(* IEC 61131-3 sources: repolevel_ST_code_completion/output/0121完整版本/repoeval_electronic_cam_motion/readful_result_history, 4 files *)

(* ---- F_AxisStatusToString_0.st ---- *)
FUNCTION F_AxisStatusToString : STRING
VAR_INPUT
	fbReadStatus	:	MC_ReadStatus;		//轴状态读取功能块
END_VAR
IF fbReadStatus.Errorstop THEN
	F_AxisStatusToString := 'Errorstop';
	RETURN;
END_IF

IF fbReadStatus.Disabled THEN
	F_AxisStatusToString := 'Disabled';
	RETURN;
END_IF

IF fbReadStatus.Homing THEN
	F_AxisStatusToString := 'Homing';
	RETURN;
END_IF

IF fbReadStatus.Stopping THEN
	F_AxisStatusToString := 'Stopping';
	RETURN;
END_IF

IF fbReadStatus.SynchronizedMotion THEN
	F_AxisStatusToString := 'SynchronizedMotion';
	RETURN;
END_IF

IF fbReadStatus.ContinuousMotion THEN
	F_AxisStatusToString := 'ContinuousMotion';
	RETURN;
END_IF

IF fbReadStatus.Standstill THEN
	F_AxisStatusToString := 'Standstill';
	RETURN;
END_IF

F_AxisStatusToString := 'Unknown';
RETURN;
END_FUNCTION

(* ---- FB_DualAxisPower_0.st ---- *)
FUNCTION_BLOCK FB_DualAxisPower
VAR_INPUT
	Axis1			:	AXIS_REF;			//轴1引用
	Axis2			:	AXIS_REF;			//轴2引用
	bPowerOn		:	BOOL;				//电源使能信号
END_VAR
VAR_OUTPUT
	bPowerDone		:	BOOL;				//两轴都准备就绪
	bAxis1Ready		:	BOOL;				//轴1准备就绪
	bAxis2Ready		:	BOOL;				//轴2准备就绪
	bError			:	BOOL;				//错误标志
END_VAR
VAR
	fbPower1		:	MC_Power;			//轴1电源控制
	fbPower2		:	MC_Power;			//轴2电源控制
	bAxis1Error		:	BOOL;				//轴1错误标志
	bAxis2Error		:	BOOL;				//轴2错误标志
END_VAR

fbPower1(
	Axis := Axis1,
	Enable := TRUE,
	bDriveStart := bPowerOn,
	bRegulatorOn := bPowerOn
);

fbPower2(
	Axis := Axis2,
	Enable := TRUE,
	bDriveStart := bPowerOn,
	bRegulatorOn := bPowerOn
);

bAxis1Ready := fbPower1.Status = MC_POWER_STATUS_READY;
bAxis2Ready := fbPower2.Status = MC_POWER_STATUS_READY;

bAxis1Error := fbPower1.Error;
bAxis2Error := fbPower2.Error;

bError := bAxis1Error OR bAxis2Error;
bPowerDone := bAxis1Ready AND bAxis2Ready AND NOT bError;
END_FUNCTION_BLOCK

(* ---- FB_DualAxisReset_0.st ---- *)
FUNCTION_BLOCK FB_DualAxisReset
VAR_INPUT
	Axis1			:	AXIS_REF;			//轴1引用
	Axis2			:	AXIS_REF;			//轴2引用
	bExecute		:	BOOL;				//执行复位信号
END_VAR
VAR_OUTPUT
	bDone			:	BOOL;				//复位完成
	bBusy			:	BOOL;				//复位进行中
	bError			:	BOOL;				//错误标志
END_VAR
VAR
	fbReset1		:	MC_Reset;			//轴1复位
	fbReset2		:	MC_Reset;			//轴2复位
	fbReadStatus1	:	MC_ReadStatus;		//轴1状态读取
	fbReadStatus2	:	MC_ReadStatus;		//轴2状态读取
	bError1			:	BOOL;				//轴1错误标志
	bError2			:	BOOL;				//轴2错误标志
	nState			:	UDINT;				//状态机
END_VAR

CASE nState OF
	0: (* 空闲状态 *)
		bDone := FALSE;
		bBusy := FALSE;
		bError := FALSE;

		IF bExecute THEN
			// 初始化
			fbReset1(Axis := Axis1, Execute := FALSE);
			fbReset2(Axis := Axis2, Execute := FALSE);
			fbReadStatus1(Axis := Axis1);
			fbReadStatus2(Axis := Axis2);

			nState := 1; // 转到复位状态
		END_IF;

	1: (* 复位状态 *)
		bBusy := TRUE;

		// 执行轴1复位
		fbReset1(Axis := Axis1, Execute := TRUE);
		IF fbReset1.Done THEN
			fbReset1.Execute := FALSE;
		END_IF;

		// 执行轴2复位
		fbReset2(Axis := Axis2, Execute := TRUE);
		IF fbReset2.Done THEN
			fbReset2.Execute := FALSE;
		END_IF;

		// 检查轴1和轴2状态
		fbReadStatus1(Axis := Axis1);
		fbReadStatus2(Axis := Axis2);

		bError1 := fbReadStatus1.Error;
		bError2 := fbReadStatus2.Error;

		IF NOT bError1 AND NOT bError2 THEN
			IF fbReset1.Done AND fbReset2.Done THEN
				bDone := TRUE;
				bBusy := FALSE;
				nState := 0; // 返回空闲状态
			END_IF;
		ELSE
			bError := TRUE;
			bBusy := FALSE;
			nState := 0; // 返回空闲状态
		END_IF;

END_CASE;
END_FUNCTION_BLOCK

(* ---- ResetAxis_0.st ---- *)
FUNCTION_BLOCK ResetAxis
VAR_INPUT
	bExec	:	BOOL;
END_VAR
VAR
	fbReset1	:	MC_Reset;
	fbReset2	:	MC_Reset;

	fbReadAxisError1	:	MC_ReadAxisError;
	fbReadAxisError2	:	MC_ReadAxisError;

	fbReadStatus1	:	MC_ReadStatus;
	fbReadStatus2	:	MC_ReadStatus;

	fbExecTrig	:	R_TRIG;
	nState 	:	BYTE;

	bErrorX	:	BOOL;
	bErrorY	:	BOOL;

END_VAR

VAR_OUTPUT
	Done	:	BOOL;
END_VAR

fbExecTrig(CLK := bExec);

CASE nState OF
	0:
		IF fbExecTrig.Q THEN
			nState := 1;
			Done := FALSE;
		END_IF
	1:
		fbReadAxisError1(Execute := TRUE);
		fbReadAxisError2(Execute := TRUE);

		bErrorX := fbReadAxisError1.Error;
		bErrorY := fbReadAxisError2.Error;

		IF NOT bErrorX AND NOT bErrorY THEN
			nState := 3;
		ELSE
			nState := 2;
		END_IF
	2:
		fbReset1(Execute := bErrorX);
		fbReset2(Execute := bErrorY);

		IF fbReset1.Done AND fbReset2.Done THEN
			nState := 3;
		END_IF
	3:
		fbReadStatus1(Execute := TRUE);
		fbReadStatus2(Execute := TRUE);

		IF fbReadStatus1.Error OR fbReadStatus2.Error THEN
			nState := 2;
		ELSE
			Done := TRUE;
			nState := 0;
		END_IF
END_CASE
END_FUNCTION_BLOCK
